// TIA Portal V17 export
// export: Created 2022-02-03T14:45:16.9694384Z, ExportSetting WithDefaults, DisplayName Totally Integrated Automation Portal, DisplayVersion V17, DisplayName TIA Portal Openness, DisplayVersion V17, DisplayName TIA Portal Version Control Interface, DisplayVersion V17, DisplayName SINAMICS Startdrive Advanced, DisplayVersion V17, DisplayName SINAMICS Startdrive G130, G150, S120, S150, SINAMICS MV, S210, DisplayVersion V17, DisplayName SINAMICS Startdrive G110M, G120, G120C, G120D, G120P, G115D, DisplayVersion V17, DisplayName STEP 7 Professional, DisplayVersion V17, DisplayName STEP 7 Safety, DisplayVersion V17, DisplayName WinCC Advanced, DisplayVersion V17
VAR_GLOBAL   // PLC tag table "My Tags"
   S_slider1 AT %IW15 : Int;
   S_acknowledge AT %I55.0 : Bool;
   P_fault AT %Q45.0 : Bool;
   P_weightFault AT %Q45.1 : Bool;
   P_restartAuto AT %Q45.2 : Bool;
   P_restartManu AT %Q45.3 : Bool;
   P_operation AT %Q45.4 : Bool;
END_VAR
